PROGRAM MAIN
VAR
END_VAR

END_PROGRAM

(* stored: Version 1.1.0.1
   POU MAIN: Id {23fff007-8416-4519-8dc4-d505da3e87b3} *)
